# EPICS substitutions: iocs/MC03/db/SAI_Global.substitutions
file /opt/epics/modules/SAI/db/SAI_Global.db {
pattern {	ASYNPORT,	TMOT,		SCAN,		P,	R,	T,	NAME,	A1,	A2,	A3,	A4,	A5,	A6,	A7,	A8}
        { 	"pmac",		"1",		".2 second",	"XF:06BMA-OP",	"{Slt:01-Ax:",	"{Slt:01}",	"InFlange Slits 01",	"O}Mtr",	"I}Mtr",	"T}Mtr",	"B}Mtr",	"DummyO}Mtr",	"DummyI}Mtr",	"DummyT}Mtr",	"DummyB}Mtr"}
}
#EOF
